INTERFACE I_CalcFocalLengthLensSet EXTENDS I_Fallible


METHOD Calculate
VAR_INPUT
    LensSet : I_LensSet;
END_VAR
VAR_IN_OUT
    FocalLength : FB_QuantityLREALPublic(Units := 'm');
END_VAR
END_METHOD

END_INTERFACE

(* stored: Version 1.1.0.1
   Itf I_CalcFocalLengthLensSet: Id {a3bee5e8-81aa-4cb0-8342-b3925dda85b9}
   Method Calculate: Id {c3aa6e0a-ee96-4697-8336-4b3722043c3b} *)
